// Error handler interface for centralised error management
INTERFACE I_ErrorHandler

METHOD AddError : BOOL
VAR_INPUT
    nCode       : UDINT;
    eSeverity   : E_Severity;
    sMessage    : STRING(255);
    sSource     : STRING(80);
END_VAR
END_METHOD

METHOD ClearErrors : BOOL
VAR_INPUT
END_VAR
END_METHOD

METHOD HasErrors : BOOL
VAR_INPUT
END_VAR
END_METHOD

METHOD HasFatal : BOOL
VAR_INPUT
END_VAR
END_METHOD

METHOD GetError : ST_ErrorInfo
VAR_INPUT
    nIndex : UDINT; // 0 = most recent
END_VAR
END_METHOD

METHOD GetCount : UDINT
VAR_INPUT
END_VAR
END_METHOD

END_INTERFACE

(* stored: Version 1.1.0.1, ProductVersion 3.1.4024.12
   Itf I_ErrorHandler: Id {C33F4C5A-8249-4BD8-9C15-3B6D08BBE5CC}
   Method AddError: Id {FD059066-C89B-43BC-9822-CBF01243CC9C}
   Method ClearErrors: Id {6E2ED222-D004-4BA9-A419-E0C00512E970}
   Method HasErrors: Id {B80923A1-EACE-4688-82E6-10E915CDB62E}
   Method HasFatal: Id {54C2AE2C-F28A-40AD-B136-485534B4830F}
   Method GetError: Id {BCBA1513-DD46-4B40-A616-C661CB72B3BD}
   Method GetCount: Id {F3ADEF9E-3EB3-4174-8358-AA6CA6D18C51} *)
